TYPE HMI_STS_LayerScan :
STRUCT
	// ErrorId:UDINT;				//Error id
END_STRUCT
END_TYPE

(* stored: Version 1.1.0.1
   DUT HMI_STS_LayerScan: Id {64e3cfaf-d06e-4d9d-ac50-2c9483b24559} *)
